PROGRAM LD_Logic
VAR
END_VAR

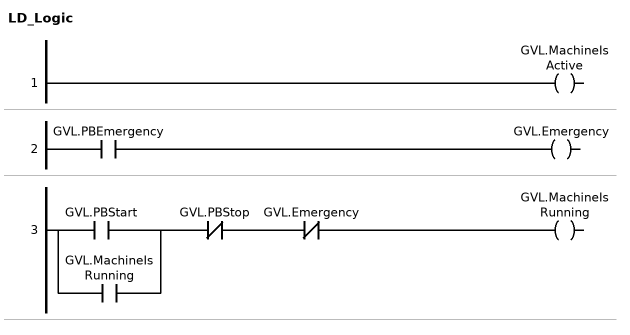
// NETWORK 1
GVL.MachineIsActive := TRUE;

// NETWORK 2
GVL.Emergency := GVL.PBEmergency;

// NETWORK 3
GVL.MachineIsRunning := (GVL.PBStart OR GVL.MachineIsRunning) AND NOT GVL.PBStop AND NOT GVL.Emergency;

END_PROGRAM

(* stored: Version 1.1.0.1, ProductVersion 3.1.4024.12
   POU LD_Logic: Id {39b509b7-7932-4c19-a752-b9e09dbae532}, SpecialFunc None *)
